(* IEC 61131-3 sources: wago750-881/, 2 files *)

(* ---- globalvar.st ---- *)
(* ========================================================================== *)
(* GLOBALE KONSTANTEN                                                         *)
(* ========================================================================== *)
VAR_GLOBAL CONSTANT
    (* Heizkreis-Pumpe Reason Bits *)
    HK_REASON_FROSTSCHUTZ    : BYTE := 16#01;
    HK_REASON_WAERMEBEDARF   : BYTE := 16#02;
    HK_REASON_OVERRIDE       : BYTE := 16#04;

    (* Brunnenpumpe Reason Bits *)
    BR_REASON_HK_ACTIVE      : BYTE := 16#01;

    (* Sollwerte *)
    CONST_VL_SOLL_MIN : REAL := 45.0;

    (* NTC Boiler Kalibrierung *)
    NTC_BOILER_A : REAL := 40536.0;
    NTC_BOILER_B : REAL := 303.1;

    (* NTC Solar Kalibrierung *)
    NTC_SOLAR_A : REAL := 26402.0;
    NTC_SOLAR_B : REAL := 60.0;

    (* VERSION *)
    VERSION_MAJOR : BYTE := 6;
    VERSION_MINOR : BYTE := 5;
    VERSION_PATCH : BYTE := 2;
END_VAR

(* ========================================================================== *)
(* GLOBALE VARIABLEN                                                          *)
(* ========================================================================== *)
VAR_GLOBAL
    (* ====================================================================== *)
    (* PHYSIKALISCHE HARDWARE                                                 *)
    (* ====================================================================== *)
    analog0 AT %IW0 : WORD;
    analog1 AT %IW1 : WORD;
    analog2 AT %IW2 : WORD;
    analog3 AT %IW3 : WORD;
    DI8chan AT %IW4 : WORD;

    Output_0      AT %QX0.0 : BOOL;
    O1_WWPump     AT %QX0.1 : BOOL;
    O2_UmwaelzHK1 AT %QX0.2 : BOOL;
    O3_Brunnen    AT %QX0.3 : BOOL;
    O5            AT %QX0.5 : BOOL;

    (* ====================================================================== *)
    (* SAMPLE & HOLD SPEICHER                                                 *)
    (* ====================================================================== *)
    S_Vorlauf    : WORD;
    S_Aussen     : WORD;
    S_Innen      : WORD;
    S_Kessel     : WORD;
    S_Warmw      : WORD;
    S_Oeltank    : WORD;
    S_Ruecklauf  : WORD;
    S_Solar      : WORD;

    (* ====================================================================== *)
    (* BERECHNETE WERTE                                                       *)
    (* ====================================================================== *)
    (* Temperaturen *)
    temp_vorlauf   : REAL;
    temp_kessel    : REAL;
    temp_aussen    : REAL;
    temp_innen     : REAL;
    temp_ruecklauf : REAL;
    temp_warmw     : REAL;
    temp_solar     : REAL;
    temp_diff_ww   : REAL;

    (* Hilfsvariablen für Sensorberechnung *)
    ohm_vorlauf   : REAL;
    ohm_kessel    : REAL;
    ohm_aussen    : REAL;
    ohm_innen     : REAL;
    ohm_ruecklauf : REAL;
    raw_warmw_real : REAL;
    raw_solar_real : REAL;

    (* PT1000 Kalibrierung *)
    PT1000_R0  : REAL := 1000.0;
    R_Mess     : REAL := 10000.0;
    U_Vers     : REAL := 24.0;
    U_SPS      : REAL := 10.0;
    Raw_Max    : REAL := 32767.0;
    U_PT       : REAL;

    (* ====================================================================== *)
    (* STEUERUNG                                                              *)
    (* ====================================================================== *)
    bSensorError      : BOOL := FALSE;
    bNachtAbsenkung   : BOOL := FALSE;
    bDataReady        : BOOL := FALSE;
    mux_state         : BOOL := FALSE;

    (* Reason Bytes *)
    bWW_Reason : BYTE := 0;
    bHK_Reason : BYTE := 0;
    bBR_Reason : BYTE := 0;

    (* Enable/Manual Signale für Pumpen *)
    bWW_Enable : BOOL := FALSE;
    bHK_Enable : BOOL := FALSE;
    bBR_Enable : BOOL := FALSE;

    bWW_Manual : BOOL := FALSE;
    bHK_Manual : BOOL := FALSE;
    bBR_Manual : BOOL := FALSE;

    (* Echtzeituhr *)
    rtc_dt      : DT;
    hour_of_day : INT;

    (* Nachtabsenkungszeiten *)
    nacht_start_hour : INT := 23;
    nacht_end_hour   : INT := 4;

    (* Timer *)
    Timer_Long   : TON;
    Timer_Short  : TON;
    Timer_Settle : TON;

    (* ====================================================================== *)
    (* OSCAT BUILDING ACTUATOR_PUMP INSTANZEN                                *)
    (* ====================================================================== *)
    ACTUATOR_WW : ACTUATOR_PUMP;
    ACTUATOR_HK : ACTUATOR_PUMP;
    ACTUATOR_BR : ACTUATOR_PUMP;

    (* ====================================================================== *)
    (* BETRIEBSSTUNDEN - NON-RETAIN                                          *)
    (* ====================================================================== *)
    WW_Runtime : UDINT := 0;  (* Hundertstel-Sekunden *)
    WW_Cycles  : UDINT := 0;  (* Anzahl Starts *)
    HK_Runtime : UDINT := 0;
    HK_Cycles  : UDINT := 0;
    BR_Runtime : UDINT := 0;
    BR_Cycles  : UDINT := 0;

    (* ====================================================================== *)
    (* MODBUS-REGISTER - MEMORY MAPPING                                      *)
    (* ====================================================================== *)
    (* WICHTIG: Modbus-Adresse = CODESYS MW-Nummer + 12288                   *)
    (*                                                                        *)
    (* Beispiel: MW32 = Modbus-Adresse 12320                                 *)
    (*           MW96 = Modbus-Adresse 12384                                 *)
    (* ====================================================================== *)

    (* MW0-31: Basis-Zähler (deprecated, für Kompatibilität) *)
    xNewVar7 AT %MW0 : ARRAY [1..16] OF INT;
    (* [1] = Zaehler_kWh (deprecated)
       [2] = Zaehler_Pumpe (deprecated)
       [3] = Zaehler_Brunnen (deprecated)
       [4-16] = Reserve *)

    (* ====================================================================== *)
    (* MW32-63: MESSWERTE & STATUS (Modbus 12320-12351)                      *)
    (* ====================================================================== *)
    xMeasure AT %MW32 : ARRAY [1..32] OF INT;
    (* [1]  = MW32  = 12320 = S_Vorlauf (Raw WORD)
       [2]  = MW33  = 12321 = S_Aussen (Raw WORD)
       [3]  = MW34  = 12322 = S_Innen (Raw WORD)
       [4]  = MW35  = 12323 = S_Kessel (Raw WORD)
       [5]  = MW36  = 12324 = S_Warmw (Raw WORD)
       [6]  = MW37  = 12325 = S_Oeltank (Raw WORD)
       [7]  = MW38  = 12326 = S_Ruecklauf (Raw WORD)
       [8]  = MW39  = 12327 = S_Solar (Raw WORD)
       [9]  = MW40  = 12328 = DI8chan (Raw WORD)
       [10] = MW41  = 12329 = hour_of_day (INT 0-23)
       [11] = MW42  = 12330 = Status-Word (INT Bitmaske)
            Bit 0: O1_WWPump aktiv
            Bit 1: O2_UmwaelzHK1 aktiv
            Bit 2: O3_Brunnen aktiv
            Bit 3: bNachtAbsenkung aktiv
            Bit 4: mux_state (Phase A/B)
            Bit 5: bDataReady
            Bit 6: bSensorError
       [12] = MW43  = 12331 = temp_diff_ww * 100 (INT, z.B. 1087 = 10.87°C)
       [13] = MW44  = 12332 = temp_kessel * 100 (INT)
       [14] = MW45  = 12333 = temp_warmw * 100 (INT)
       [15] = MW46  = 12334 = temp_vorlauf * 100 (INT)
       [16] = MW47  = 12335 = VERSION (Byte-Packed: High=Major, Low=Minor)
       [17] = MW48  = 12336 = VERSION_PATCH (INT)
       [18] = MW49  = 12337 = Seriennummer (INT, fixiert auf 15)
       [19] = MW50  = 12338 = WW_Runtime in Sekunden (INT, max 32767s)
       [20] = MW51  = 12339 = HK_Runtime in Sekunden (INT, max 32767s)
       [21] = MW52  = 12340 = BR_Runtime in Sekunden (INT, max 32767s)
       [22] = MW53  = 12341 = WW_Cycles (INT, Anzahl Starts)
       [23] = MW54  = 12342 = HK_Cycles (INT, Anzahl Starts)
       [24] = MW55  = 12343 = BR_Cycles (INT, Anzahl Starts)
       [25] = MW56  = 12344 = bWW_Reason (INT, Low-Byte = Bitmaske)
       [26] = MW57  = 12345 = bHK_Reason (INT, Low-Byte = Bitmaske)
       [27] = MW58  = 12346 = bBR_Reason (INT, Low-Byte = Bitmaske)
       [28] = MW59  = 12347 = temp_aussen * 100 (INT)
       [29] = MW60  = 12348 = temp_innen * 100 (INT)
       [30] = MW61  = 12349 = temp_ruecklauf * 100 (INT)
       [31] = MW62  = 12350 = temp_solar * 100 (INT)
       [32] = MW63  = 12351 = QB0 Physical Output Byte (INT) *)

    (* ====================================================================== *)
    (* MW96-111: SETPOINTS & KONFIGURATION (Modbus 12384-12399)              *)
    (* ====================================================================== *)
    xSetpoints AT %MW96 : ARRAY [1..16] OF INT;
    (* [1]  = MW96  = 12384 = Soll-Temperatur Vorlauf * 100 (4500 = 45.0°C)
       [2]  = MW97  = 12385 = Soll-Temperatur Warmwasser * 100
       [3]  = MW98  = 12386 = Hysterese Vorlauf * 100
       [4]  = MW99  = 12387 = Hysterese Warmwasser * 100
       [5]  = MW100 = 12388 = Nachtabsenkung Start (Stunde 0-23, -1=nicht gesetzt)
       [6]  = MW101 = 12389 = Nachtabsenkung Ende (Stunde 0-23, -1=nicht gesetzt)
       [7]  = MW102 = 12390 = Nachtabsenkung Temperatur * 100
       [8]  = MW103 = 12391 = Multiplexer Zeit Phase A (Sekunden)
       [9]  = MW104 = 12392 = Multiplexer Zeit Phase B (Sekunden)
       [10] = MW105 = 12393 = Frostschutz-Schwelle * 100 (-1300 = -13.0°C, 0=nicht gesetzt)
       [11] = MW106 = 12394 = Max Vorlauf * 100
       [12] = MW107 = 12395 = Pumpen Nachlaufzeit (Sekunden)
       [13] = MW108 = 12396 = HeatPump R290 Watertank Temp * 100 (von Python geschrieben)
       [14] = MW109 = 12397 = Pumpen-Override WW (-1=Force OFF, 0=Auto, 1=Force ON)
       [15] = MW110 = 12398 = Pumpen-Override HK (-1=Force OFF, 0=Auto, 1=Force ON)
       [16] = MW111 = 12399 = Pumpen-Override Brunnen (-1=Force OFF, 0=Auto, 1=Force ON) *)

    (* ====================================================================== *)
    (* MW128-135: SYSTEM-DIAGNOSE (Modbus 12416-12423)                       *)
    (* ====================================================================== *)
    xSystem AT %MW128 : ARRAY [1..8] OF INT;
    (* [1] = MW128 = 12416 = Uptime Sekunden (low word, 0-65535)
       [2] = MW129 = 12417 = Uptime Sekunden (high word) ? 32-bit kombiniert
       [3] = MW130 = 12418 = Fehler-Counter
       [4] = MW131 = 12419 = CPU Load %
       [5] = MW132 = 12420 = Cycle time min (ms)
       [6] = MW133 = 12421 = Cycle time max (ms)
       [7] = MW134 = 12422 = Cycle time avg (ms)
       [8] = MW135 = 12423 = Reserve *)

    (* ====================================================================== *)
    (* MW144-151: ALARM-REGISTER (Modbus 12432-12439)                        *)
    (* ====================================================================== *)
    xAlarms AT %MW144 : ARRAY [1..8] OF INT;
    (* [1] = MW144 = 12432 = Alarm-Bitmaske
            Bit 0: Sensor Vorlauf Fehler
            Bit 1: Sensor Aussen Fehler
            Bit 2: Sensor Kessel Fehler
            Bit 3: Sensor WW Fehler
            Bit 4-15: Reserve
       [2] = MW145 = 12433 = Fehler-Counter Sensor Vorlauf
       [3] = MW146 = 12434 = Fehler-Counter Sensor Aussen
       [4] = MW147 = 12435 = Fehler-Counter Sensor Kessel
       [5] = MW148 = 12436 = Fehler-Counter Sensor WW
       [6-8] = Reserve *)

    (* ====================================================================== *)
    (* MW160-167: STATISTIK (Modbus 12448-12455)                             *)
    (* ====================================================================== *)
    xStats AT %MW160 : ARRAY [1..8] OF INT;
    (* [1] = MW160 = 12448 = Betriebsstunden HK (Stunden)
       [2] = MW161 = 12449 = Betriebsstunden WW (Stunden)
       [3] = MW162 = 12450 = Betriebsstunden BR (Stunden)
       [4] = MW163 = 12451 = Starts HK
       [5] = MW164 = 12452 = Starts WW
       [6] = MW165 = 12453 = Starts BR
       [7] = MW166 = 12454 = Reserve
       [8] = MW167 = 12455 = Reserve *)

    (* ====================================================================== *)
    (* HILFSVARIABLEN                                                         *)
    (* ====================================================================== *)
    uptime_seconds : UDINT := 0;
    error_counter : INT := 0;
    QB0_shadow : BYTE;  (* Kopie von %QB0 für Modbus *)
END_VAR

(* ========================================================================== *)
(* REGISTER-MAPPING ZUSAMMENFASSUNG                                          *)
(* ========================================================================== *)
(*
WICHTIGE ADRESSEN FÜR PYTHON:

Stunden-Setpoint schreiben:
  MW0 = 12288 (hour_of_day wird von Python geschrieben)

Messwerte lesen:
  MW32-63 = 12320-12351 (xMeasure[1..32])

Setpoints schreiben:
  MW96-111 = 12384-12399 (xSetpoints[1..16])

  Wichtigste:
    MW100 = 12388 = Nachtabsenkung Start
    MW101 = 12389 = Nachtabsenkung Ende
    MW105 = 12393 = Frostschutz-Schwelle
    MW108 = 12396 = R290 Wassertank Temp
    MW109 = 12397 = WW Override
    MW110 = 12398 = HK Override
    MW111 = 12399 = BR Override

Physical Outputs lesen:
  %QB0 = 512 (Physical Output Byte)

System-Info lesen:
  MW128-135 = 12416-12423 (xSystem[1..8])
*)

(* ---- heizung.st ---- *)
(* ========================================================================== *)
(* PLC_PRG - HAUPTPROGRAMM v6.5.2                                            *)
(* ========================================================================== *)

(* Initialisierung *)
bWW_Reason := 0;
bHK_Reason := 0;
bBR_Reason := 0;
xAlarms[1] := 0;

(* ========================================================================== *)
(* 1. ECHTZEITUHR & NACHTABSENKUNG - DYNAMISCH                              *)
(* ========================================================================== *)
rtc_dt := SysRtcGetTime(TRUE);
hour_of_day := DWORD_TO_INT((DT_TO_DWORD(rtc_dt) / 3600) MOD 24);

(* Nachtabsenkungszeiten aus xSetpoints[5] und [6] lesen *)
IF (xSetpoints[5] < 0) OR (xSetpoints[5] > 23) OR (xSetpoints[6] < 0) OR (xSetpoints[6] > 23) THEN
    (* Ungültige Werte -> DEAKTIVIERT *)
    bNachtAbsenkung := FALSE;
ELSIF (xSetpoints[5] = 0) AND (xSetpoints[6] = 0) THEN
    (* Beide 0 = nicht initialisiert -> DEAKTIVIERT *)
    bNachtAbsenkung := FALSE;
ELSE
    (* Gültige Werte übernehmen *)
    nacht_start_hour := xSetpoints[5];
    nacht_end_hour := xSetpoints[6];

    (* Nachtabsenkung berechnen *)
    IF nacht_start_hour < nacht_end_hour THEN
        (* Normal: z.B. 6-10 Uhr *)
        bNachtAbsenkung := (hour_of_day >= nacht_start_hour) AND (hour_of_day < nacht_end_hour);
    ELSE
        (* Über Mitternacht: z.B. 23-4 Uhr *)
        bNachtAbsenkung := (hour_of_day >= nacht_start_hour) OR (hour_of_day < nacht_end_hour);
    END_IF;
END_IF;

(* ========================================================================== *)
(* 2. MULTIPLEXER                                                             *)
(* ========================================================================== *)
IF mux_state THEN
    Timer_Long(IN := TRUE, PT := T#51S);
    IF Timer_Long.Q THEN
        mux_state := FALSE;
        Timer_Long(IN := FALSE);
        Timer_Settle(IN := FALSE);
    END_IF;
ELSE
    Timer_Short(IN := TRUE, PT := T#8S);
    IF Timer_Short.Q THEN
        mux_state := TRUE;
        Timer_Short(IN := FALSE);
        Timer_Settle(IN := FALSE);
    END_IF;
END_IF;

Output_0 := mux_state;
Timer_Settle(IN := TRUE, PT := T#2S);
bDataReady := Timer_Settle.Q;

(* ========================================================================== *)
(* 3. SAMPLE & HOLD                                                           *)
(* ========================================================================== *)
IF bDataReady THEN
    IF mux_state THEN
        S_Vorlauf := analog0;
        S_Aussen  := analog1;
        S_Innen   := analog2;
        S_Kessel  := analog3;
    ELSE
        S_Warmw     := analog0;
        S_Oeltank   := analog1;
        S_Ruecklauf := analog2;
        S_Solar     := analog3;
    END_IF;
END_IF;

(* ========================================================================== *)
(* 4. TEMPERATUR-BERECHNUNGEN                                                 *)
(* ========================================================================== *)
U_PT := (WORD_TO_REAL(S_Vorlauf) / Raw_Max) * U_SPS;
ohm_vorlauf := (U_PT * R_Mess) / (U_Vers - U_PT);
temp_vorlauf := TEMP_PT(ohm_vorlauf, PT1000_R0);

U_PT := (WORD_TO_REAL(S_Kessel) / Raw_Max) * U_SPS;
ohm_kessel := (U_PT * R_Mess) / (U_Vers - U_PT);
temp_kessel := TEMP_PT(ohm_kessel, PT1000_R0);

U_PT := (WORD_TO_REAL(S_Aussen) / Raw_Max) * U_SPS;
ohm_aussen := (U_PT * R_Mess) / (U_Vers - U_PT);
temp_aussen := TEMP_PT(ohm_aussen, PT1000_R0);

U_PT := (WORD_TO_REAL(S_Innen) / Raw_Max) * U_SPS;
ohm_innen := (U_PT * R_Mess) / (U_Vers - U_PT);
temp_innen := TEMP_PT(ohm_innen, PT1000_R0);

U_PT := (WORD_TO_REAL(S_Ruecklauf) / Raw_Max) * U_SPS;
ohm_ruecklauf := (U_PT * R_Mess) / (U_Vers - U_PT);
temp_ruecklauf := TEMP_PT(ohm_ruecklauf, PT1000_R0);

raw_warmw_real := WORD_TO_REAL(S_Warmw);
IF (raw_warmw_real >= 4000.0) AND (raw_warmw_real <= 45000.0) THEN
    temp_warmw := (NTC_BOILER_A - raw_warmw_real) / NTC_BOILER_B;
ELSE
    temp_warmw := 0.0;
END_IF;

raw_solar_real := WORD_TO_REAL(S_Solar);
IF (raw_solar_real >= 4000.0) AND (raw_solar_real <= 40000.0) THEN
    temp_solar := (raw_solar_real - NTC_SOLAR_A) / NTC_SOLAR_B;
ELSE
    temp_solar := 0.0;
END_IF;

temp_diff_ww := temp_kessel - temp_warmw;
bSensorError := FALSE;

(* ========================================================================== *)
(* 5. PUMPENSTEUERUNG - MIT INVERTIERTER RELAIS-LOGIK                       *)
(* ========================================================================== *)
watertank_waschk := xSetpoints[13];

(* ========================================================================== *)
(* 5.1 WARMWASSER-PUMPE - IGNORIERT NACHTABSENKUNG!                         *)
(* ========================================================================== *)
bWW_Reason := BYTE#0;

(* Temperaturdifferenz - OHNE Nachtabsenkungsprüfung *)
IF temp_diff_ww >= 2.0 THEN
    bWW_Reason := BYTE#1;  (* WW_REASON_TEMP_DIFF *)
END_IF;

(* Override-Handling *)
IF xSetpoints[14] < INT#0 THEN
    bWW_Enable := FALSE;
    bWW_Manual := TRUE;
    bWW_Reason := BYTE#0;
ELSIF xSetpoints[14] > INT#0 THEN
    bWW_Enable := TRUE;
    bWW_Manual := TRUE;
    bWW_Reason := BYTE#4;  (* WW_REASON_OVERRIDE *)
ELSE
    bWW_Enable := (bWW_Reason > BYTE#0);
    bWW_Manual := FALSE;
END_IF;

ACTUATOR_WW(
    IN := bWW_Enable,
    MANUAL := bWW_Manual,
    RST := FALSE,
    MIN_ONTIME := T#120S,
    MIN_OFFTIME := T#60S,
    RUN_EVERY := T#10000M,
    RUNTIME := WW_Runtime,
    CYCLES := WW_Cycles
);

(* Invertierte Relais-Logik *)
IF xSetpoints[14] < INT#0 THEN
    O1_WWPump := NOT FALSE;
ELSIF xSetpoints[14] > INT#0 THEN
    O1_WWPump := NOT TRUE;
ELSE
    O1_WWPump := NOT ACTUATOR_WW.PUMP;
END_IF;

(* ========================================================================== *)
(* 5.2 HEIZKREIS-PUMPE - BEACHTET NACHTABSENKUNG                            *)
(* ========================================================================== *)
bHK_Reason := BYTE#0;

(* Frostschutz - dynamisch aus xSetpoints[10] *)
IF xSetpoints[10] <> 0 THEN
    IF temp_aussen < (INT_TO_REAL(xSetpoints[10]) / 100.0) THEN
        bHK_Reason := HK_REASON_FROSTSCHUTZ;
    END_IF;
END_IF;

(* Wärmebedarf nur außerhalb Nachtabsenkung *)
IF (temp_vorlauf < CONST_VL_SOLL_MIN) AND NOT bNachtAbsenkung THEN
    bHK_Reason := bHK_Reason OR HK_REASON_WAERMEBEDARF;
END_IF;

(* Override-Handling *)
IF xSetpoints[15] < INT#0 THEN
    bHK_Enable := FALSE;
    bHK_Manual := TRUE;
    bHK_Reason := BYTE#0;
ELSIF xSetpoints[15] > INT#0 THEN
    bHK_Enable := TRUE;
    bHK_Manual := TRUE;
    bHK_Reason := bHK_Reason OR HK_REASON_OVERRIDE;
ELSE
    bHK_Enable := (bHK_Reason > BYTE#0);
    bHK_Manual := FALSE;
END_IF;

ACTUATOR_HK(
    IN := bHK_Enable,
    MANUAL := bHK_Manual,
    RST := FALSE,
    MIN_ONTIME := T#5M,
    MIN_OFFTIME := T#2M,
    RUN_EVERY := T#10000M,
    RUNTIME := HK_Runtime,
    CYCLES := HK_Cycles
);

(* Invertierte Relais-Logik *)
IF xSetpoints[15] < INT#0 THEN
    O2_UmwaelzHK1 := NOT FALSE;
ELSIF xSetpoints[15] > INT#0 THEN
    O2_UmwaelzHK1 := NOT TRUE;
ELSE
    O2_UmwaelzHK1 := NOT ACTUATOR_HK.PUMP;
END_IF;
(* ========================================================================== *)
(* 5.3 BRUNNENPUMPE - LÄUFT IMMER (außer Force OFF)                         *)
(* ========================================================================== *)
bBR_Reason := BR_REASON_HK_ACTIVE;  (* Immer gesetzt = läuft immer *)

(* Override-Handling *)
IF xSetpoints[16] < INT#0 THEN
    (* Force OFF *)
    O3_Brunnen := FALSE;
    bBR_Reason := BYTE#0;
ELSIF xSetpoints[16] > INT#0 THEN
    (* Force ON *)
    O3_Brunnen := TRUE;
    bBR_Reason := BYTE#4;
ELSE
    (* Auto = IMMER AN *)
    O3_Brunnen := TRUE;
END_IF;

(* ACTUATOR nur für Runtime-Tracking *)
ACTUATOR_BR(
    IN := O3_Brunnen,
    MANUAL := FALSE,
    RST := FALSE,
    MIN_ONTIME := T#1S,
    MIN_OFFTIME := T#1S,
    RUN_EVERY := T#10000M,
    RUNTIME := BR_Runtime,
    CYCLES := BR_Cycles
);
(* ========================================================================== *)
(* 6. UPTIME & BETRIEBSSTUNDEN                                                *)
(* ========================================================================== *)
Timer_OneSecond(IN := TRUE, PT := T#1000ms);
IF Timer_OneSecond.Q THEN
    Timer_OneSecond(IN := FALSE);
    second_tick := TRUE;
    uptime_seconds := uptime_seconds + 1;
ELSE
    second_tick := FALSE;
END_IF;

(* ========================================================================== *)
(* 7. MODBUS MAPPING                                                          *)
(* ========================================================================== *)
status_word := INT#0;

(* Status-Word mit invertierten Pumpen *)
IF O1_WWPump = FALSE THEN status_word := status_word + INT#1; END_IF;
IF O2_UmwaelzHK1 = FALSE THEN status_word := status_word + INT#2; END_IF;
IF O3_Brunnen THEN status_word := status_word + INT#4; END_IF;
IF bNachtAbsenkung THEN status_word := status_word + INT#8; END_IF;
IF mux_state THEN status_word := status_word + INT#16; END_IF;
IF bDataReady THEN status_word := status_word + INT#32; END_IF;
IF bSensorError THEN status_word := status_word + INT#64; END_IF;

version_word := BYTE_TO_INT(VERSION_MAJOR) * INT#256 + BYTE_TO_INT(VERSION_MINOR);

QB0_shadow := %QB0;

(* xMeasure Array füllen *)
xMeasure[1]  := WORD_TO_INT(S_Vorlauf);
xMeasure[2]  := WORD_TO_INT(S_Aussen);
xMeasure[3]  := WORD_TO_INT(S_Innen);
xMeasure[4]  := WORD_TO_INT(S_Kessel);
xMeasure[5]  := WORD_TO_INT(S_Warmw);
xMeasure[6]  := WORD_TO_INT(S_Oeltank);
xMeasure[7]  := WORD_TO_INT(S_Ruecklauf);
xMeasure[8]  := WORD_TO_INT(S_Solar);
xMeasure[9]  := WORD_TO_INT(DI8chan);
xMeasure[10] := hour_of_day;
xMeasure[11] := status_word;

temp_var := REAL_TO_INT(temp_diff_ww * 100.0);
xMeasure[12] := temp_var;
temp_var := REAL_TO_INT(temp_kessel * 100.0);
xMeasure[13] := temp_var;
temp_var := REAL_TO_INT(temp_warmw * 100.0);
xMeasure[14] := temp_var;
temp_var := REAL_TO_INT(temp_vorlauf * 100.0);
xMeasure[15] := temp_var;

xMeasure[16] := version_word;
xMeasure[17] := BYTE_TO_INT(VERSION_PATCH);
xMeasure[18] := INT#15;

IF WW_Runtime < 32767 THEN
    xMeasure[19] := UDINT_TO_INT(WW_Runtime);
ELSE
    xMeasure[19] := 32767;
END_IF;

IF HK_Runtime < 32767 THEN
    xMeasure[20] := UDINT_TO_INT(HK_Runtime);
ELSE
    xMeasure[20] := 32767;
END_IF;

IF BR_Runtime < 32767 THEN
    xMeasure[21] := UDINT_TO_INT(BR_Runtime);
ELSE
    xMeasure[21] := 32767;
END_IF;

IF WW_Cycles < 32767 THEN
    xMeasure[22] := UDINT_TO_INT(WW_Cycles);
ELSE
    xMeasure[22] := 32767;
END_IF;

IF HK_Cycles < 32767 THEN
    xMeasure[23] := UDINT_TO_INT(HK_Cycles);
ELSE
    xMeasure[23] := 32767;
END_IF;

IF BR_Cycles < 32767 THEN
    xMeasure[24] := UDINT_TO_INT(BR_Cycles);
ELSE
    xMeasure[24] := 32767;
END_IF;

xMeasure[25] := BYTE_TO_INT(bWW_Reason);
xMeasure[26] := BYTE_TO_INT(bHK_Reason);
xMeasure[27] := BYTE_TO_INT(bBR_Reason);

temp_var := REAL_TO_INT(temp_aussen * 100.0);
xMeasure[28] := temp_var;
temp_var := REAL_TO_INT(temp_innen * 100.0);
xMeasure[29] := temp_var;
temp_var := REAL_TO_INT(temp_ruecklauf * 100.0);
xMeasure[30] := temp_var;
temp_var := REAL_TO_INT(temp_solar * 100.0);
xMeasure[31] := temp_var;

xMeasure[32] := BYTE_TO_INT(QB0_shadow);

(* xSystem Array füllen *)
xSystem[1] := UDINT_TO_INT(uptime_seconds MOD UDINT#65536);
xSystem[2] := UDINT_TO_INT(uptime_seconds / UDINT#65536);
xSystem[3] := error_counter;

(* xStats Array füllen *)
xStats[1] := UDINT_TO_INT(HK_Runtime / 3600);
xStats[2] := UDINT_TO_INT(WW_Runtime / 3600);
xStats[3] := UDINT_TO_INT(BR_Runtime / 3600);

IF HK_Cycles < 32767 THEN
    xStats[4] := UDINT_TO_INT(HK_Cycles);
ELSE
    xStats[4] := 32767;
END_IF;

IF WW_Cycles < 32767 THEN
    xStats[5] := UDINT_TO_INT(WW_Cycles);
ELSE
    xStats[5] := 32767;
END_IF;

IF BR_Cycles < 32767 THEN
    xStats[6] := UDINT_TO_INT(BR_Cycles);
ELSE
    xStats[6] := 32767;
END_IF;
